(* CODESYS project code-dry-martini.project

Project tree, tasks and I/O mapping:
  Device : CODESYS Control Win V3, 3S - Smart Software Solutions GmbH, order no. 305021, version 3.5.6.10
    application Application
      libraries: Standard, * (System)
      task MainTask (cyclic, interval t#25ms, priority 1) calls PLC_PRG, Controller
      task Secondary_Tasks (cyclic, interval t#50ms, priority 2) calls Batelada, Envase, Descartar
      task Simulacao (cyclic, interval t#100ms, priority 1) calls SimulaContadores, SimulaSensores
      task PWM (cyclic, interval t#50ms, priority 1) calls pwmpou
      program PLC_PRG [LD]
      global variables Globals
      program Batelada [SFC]: ACT1_add_gin_and_vermouth, ACT2_stop_adding_vermouth, ACT3_stop_adding_start_mixing, ACT4_stop_cooling, ACT5_stop_mixing, ACT6_close107, ACT7_finish_transfer, Step10_entry, ACT12_LSHH, ACT13_start_transfer
      program Envase [SFC]: ACT8_start_engine, ACT9_stop_and_fill, ACT10_stop_filling, ACT14_setup_timers
      program SimulaSensores [ST]
      program SimulaContadores [ST]
      program Descartar [SFC]: Step0_entry, Step1_entry, Step2_entry, Step3_entry
      program Controller [SFC]: Init_entry
      trace PWM (task MainTask): LIGA_MOTOR, M101
      program pwmpou [SFC]: ACT15_time_control, ACT16_on, ACT17_off
      Symbols
*)

// Device/Application/Globals
VAR_GLOBAL
	// ATUADORES
	FCV101: BOOL := 0;
	FCV102: BOOL := 0;
	FCV103: BOOL := 0;
	FCV104: BOOL := 0;
	FCV105: BOOL := 0;
	FCV106: BOOL := 0;
	FCV107: BOOL := 0;
	BA101: BOOL := 0;
	FCV201: BOOL := 0;
	M101: BOOL := 0;
	M201: BOOL := 0;
	
	// SENSORES
	TSL101: BOOL := 0;
	LSL101: BOOL := 0;
	LSL102: BOOL := 0;
	LSH101: BOOL := 0;
	LSH102: BOOL := 0;
	LSL201: BOOL := 0;
	FV201: BOOL := 0;
	ZY201: BOOL := 0;
	ZY202: BOOL := 0;
	LSH201: BOOL := 0;
	LSHH201: BOOL := 0;
	
	// VARIAVEIS DE CONTROLE
	LigaAux: BOOL := 0;
	Emg: BOOL := 0;
	Auto: BOOL := 0;
	TempRM01: REAL := 25;
	TempAmbienteCelsius: REAL := 25;
	CapacidadeJA01: REAL := 15;
	Alert_TR01Empty: BOOL := 0;
	LIGA_MOTOR: BOOL := 0;
	
	//CONTADORES
	FQ101: REAL := 0; 
	FQ102: REAL := 0;
	FQ103: REAL := 0;
	FQ201: REAL := 0;
	RM01: REAL := 0;
	TP01: REAL := 0;
	JA01: REAL := 0;
	nBarril: INT := 0;
	
	// TIMERS
	tZY202: REAL := 0;
	tZY201: REAL := 0;
	
	ALARM3: BOOL := FALSE;
END_VAR

// Device/Application/PLC_PRG
PROGRAM PLC_PRG
VAR
	Liga: BOOL;
	// Emg: é global
	// Auto: é global
	Man: BOOL;
END_VAR

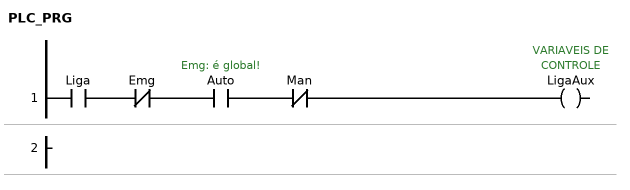
// NETWORK 1
//   Auto: Emg: é global!
//   LigaAux: VARIAVEIS DE CONTROLE
LigaAux := Liga AND NOT Emg AND Auto AND NOT Man;

// NETWORK 2

END_PROGRAM

// Device/Application/Controller
PROGRAM Controller
VAR
END_VAR

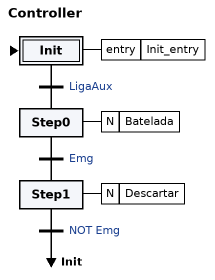
INITIAL_STEP Init:
    Init_entry(P1);  // entry action
END_STEP
TRANSITION FROM Init TO Step0
    := LigaAux;
END_TRANSITION
STEP Step0:
    Batelada(N);
END_STEP
TRANSITION FROM Step0 TO Step1
    := Emg;
END_TRANSITION
STEP Step1:
    Descartar(N);
END_STEP
TRANSITION FROM Step1 TO Init
    := NOT Emg;
END_TRANSITION

ACTION Init_entry:
TempAmbienteCelsius := 25;
CapacidadeJA01 := 15;
TempRM01:=TempAmbienteCelsius;
END_ACTION

END_PROGRAM

// Device/Application/Batelada
PROGRAM Batelada
VAR
END_VAR

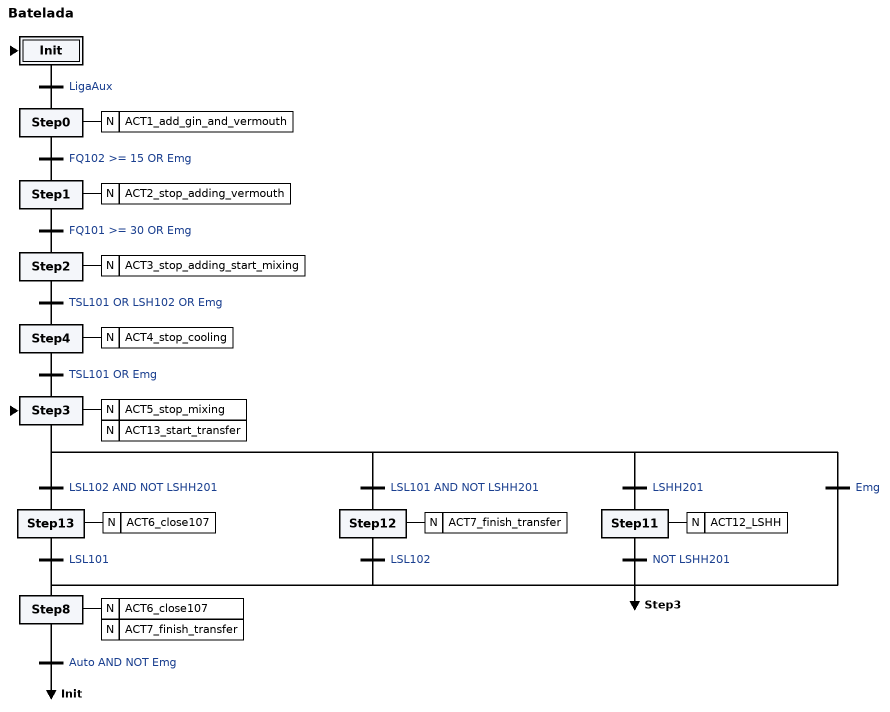
INITIAL_STEP Init:
END_STEP
TRANSITION FROM Init TO Step0
    := LigaAux;
END_TRANSITION
STEP Step0:
    ACT1_add_gin_and_vermouth(N);
END_STEP
TRANSITION FROM Step0 TO Step1
    := FQ102 >= 15 OR Emg;
END_TRANSITION
STEP Step1:
    ACT2_stop_adding_vermouth(N);
END_STEP
TRANSITION FROM Step1 TO Step2
    := FQ101 >= 30 OR Emg;
END_TRANSITION
STEP Step2:
    ACT3_stop_adding_start_mixing(N);
END_STEP
TRANSITION FROM Step2 TO Step4
    := TSL101 OR LSH102 OR Emg;
END_TRANSITION
STEP Step4:
    ACT4_stop_cooling(N);
END_STEP
TRANSITION FROM Step4 TO Step3
    := TSL101 OR Emg;
END_TRANSITION
STEP Step3:
    ACT5_stop_mixing(N);
    ACT13_start_transfer(N);
END_STEP
TRANSITION FROM Step3 TO Step13
    := LSL102 AND NOT LSHH201;
END_TRANSITION
STEP Step13:
    ACT6_close107(N);
END_STEP
TRANSITION FROM Step13 TO Step8
    := LSL101;
END_TRANSITION
TRANSITION FROM Step3 TO Step12
    := LSL101 AND NOT LSHH201;
END_TRANSITION
STEP Step12:
    ACT7_finish_transfer(N);
END_STEP
TRANSITION FROM Step12 TO Step8
    := LSL102;
END_TRANSITION
TRANSITION FROM Step3 TO Step11
    := LSHH201;
END_TRANSITION
STEP Step11:
    ACT12_LSHH(N);
END_STEP
TRANSITION FROM Step11 TO Step3
    := NOT LSHH201;
END_TRANSITION
TRANSITION FROM Step3 TO Step8
    := Emg;
END_TRANSITION
STEP Step8:
    ACT6_close107(N);
    ACT7_finish_transfer(N);
END_STEP
TRANSITION FROM Step8 TO Init
    := Auto AND NOT Emg;
END_TRANSITION

ACTION ACT1_add_gin_and_vermouth:
FCV101:=TRUE;
FCV102:=TRUE;
END_ACTION

ACTION ACT2_stop_adding_vermouth:
FCV102:=FALSE;
END_ACTION

ACTION ACT3_stop_adding_start_mixing:
FCV101:=FALSE;
LIGA_MOTOR:=TRUE;
FCV103:=TRUE;
END_ACTION

ACTION ACT4_stop_cooling:
FCV103:=FALSE;
END_ACTION

ACTION ACT5_stop_mixing:
LIGA_MOTOR:=FALSE;
END_ACTION

ACTION ACT6_close107:
FCV107:=FALSE;
END_ACTION

ACTION ACT7_finish_transfer:
FCV104:=FALSE;
FCV105:=FALSE;
BA101:=FALSE;
END_ACTION

ACTION Step10_entry:
FCV107:=TRUE;
FCV104:=TRUE;
FCV105:=TRUE;
BA101:=TRUE;
END_ACTION

ACTION ACT12_LSHH:
FCV104:=FALSE;
FCV105:=FALSE;
BA101:=FALSE;

IF TP01 <= 95 THEN
	LSHH201 := FALSE;
END_IF
END_ACTION

ACTION ACT13_start_transfer:
FCV107:=TRUE;
FCV104:=TRUE;
FCV105:=TRUE;
BA101:=TRUE;
END_ACTION

END_PROGRAM

// Device/Application/Envase
PROGRAM Envase
VAR
END_VAR

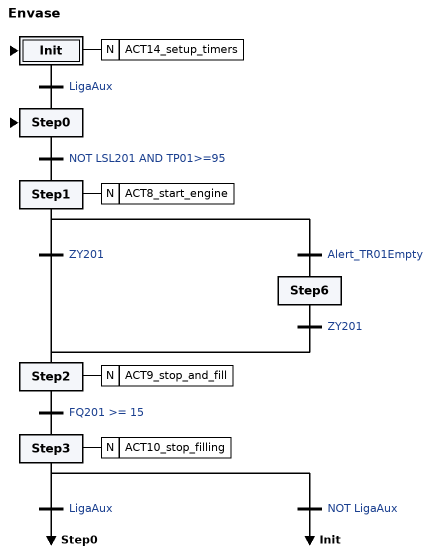
INITIAL_STEP Init:
    ACT14_setup_timers(N);
END_STEP
TRANSITION FROM Init TO Step0
    := LigaAux;
END_TRANSITION
STEP Step0:
END_STEP
TRANSITION FROM Step0 TO Step1
    := NOT LSL201 AND TP01>=95;
END_TRANSITION
STEP Step1:
    ACT8_start_engine(N);
END_STEP
TRANSITION FROM Step1 TO Step2
    := ZY201;
END_TRANSITION
TRANSITION FROM Step1 TO Step6
    := Alert_TR01Empty;
END_TRANSITION
STEP Step6:
END_STEP
TRANSITION FROM Step6 TO Step2
    := ZY201;
END_TRANSITION
STEP Step2:
    ACT9_stop_and_fill(N);
END_STEP
TRANSITION FROM Step2 TO Step3
    := FQ201 >= 15;
END_TRANSITION
STEP Step3:
    ACT10_stop_filling(N);
END_STEP
TRANSITION FROM Step3 TO Step0
    := LigaAux;
END_TRANSITION
TRANSITION FROM Step3 TO Init
    := NOT LigaAux;
END_TRANSITION

ACTION ACT8_start_engine:
M201:=TRUE;
END_ACTION

ACTION ACT9_stop_and_fill:
M201:=FALSE;
FCV201:=TRUE;
IF(Step2.t = T#15MS) THEN	
	ALARM3:=TRUE;
END_IF;
END_ACTION

ACTION ACT10_stop_filling:
FCV201:=FALSE;
END_ACTION

ACTION ACT14_setup_timers:
tZY202:=0;
tZY201:=0;
nBarril:=0;
END_ACTION

END_PROGRAM

// Device/Application/Descartar
PROGRAM Descartar
VAR
END_VAR

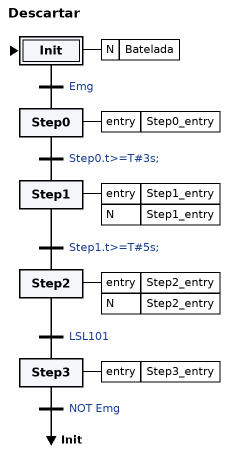
INITIAL_STEP Init:
    Batelada(N);
END_STEP
TRANSITION FROM Init TO Step0
    := Emg;
END_TRANSITION
STEP Step0:
    Step0_entry(P1);  // entry action
END_STEP
TRANSITION FROM Step0 TO Step1
    := Step0.t>=T#3s;
END_TRANSITION
STEP Step1:
    Step1_entry(P1);  // entry action
    Step1_entry(N);
END_STEP
TRANSITION FROM Step1 TO Step2
    := Step1.t>=T#5s;
END_TRANSITION
STEP Step2:
    Step2_entry(P1);  // entry action
    Step2_entry(N);
END_STEP
TRANSITION FROM Step2 TO Step3
    := LSL101;
END_TRANSITION
STEP Step3:
    Step3_entry(P1);  // entry action
END_STEP
TRANSITION FROM Step3 TO Init
    := NOT Emg;
END_TRANSITION

ACTION Step0_entry:
FCV101:=FALSE;
FCV102:=FALSE;
FCV103:=FALSE;
LIGA_MOTOR:=FALSE;
END_ACTION

ACTION Step1_entry:
FCV104:=TRUE;
FCV106:=TRUE;
BA101:=FALSE;
END_ACTION

ACTION Step2_entry:
BA101:=TRUE;
END_ACTION

ACTION Step3_entry:
BA101:=FALSE;
FCV104:=FALSE;
FCV105:=FALSE;
FCV106:=FALSE;
FCV107:=FALSE;
END_ACTION

END_PROGRAM

// Device/Application/SimulaContadores
PROGRAM SimulaContadores
VAR
	CapacidadeJaquetaRM01Litros: INT:=20; //capacidade em litros da jaqueta de resfriamento de RM01 (omisso na especificação)
	TempAmbienteCulsius: INT:= 25; //temperatura ambiente em celsius
	TOTALGIN: REAL:=0;
	TOTALVER: REAL:=0;
	TOTALDRY: REAL:=0;
//	LSL102: BOOL;
END_VAR

//ATENCAO: ESTE PROGRAMA RODA A CADA 100ms!

IF FCV101 THEN
	FQ101:=FQ101+0.6; // GIN 360 L/min = 6 L/s
	RM01:=RM01+0.6;
	TOTALGIN:=TOTALGIN+0.6;
	ELSE
		FQ101:=0;
END_IF

IF FCV102 THEN
	FQ102:=FQ102+0.5; // VERMOUTH 18 m³/h = 5 L/min
	RM01:=RM01+0.5;
	TOTALVER:=TOTALVER+0.5;
	ELSE
		FQ102:=0;
END_IF

IF FCV105 AND BA101 AND FCV104 THEN
	FQ103:=FQ103+1.5; // DRY MARTINI 54 m³/h = 15 L/min
	TP01:=TP01+1.5;
	TOTALDRY:=TOTALDRY+1.5;
ELSE
	IF NOT FCV105 THEN
		FQ103:=0;
	END_IF
END_IF

IF FCV104 AND RM01 > 0 THEN
	RM01:=RM01-1.5; 
END_IF

IF FCV201 AND TP01 > 0  THEN
	TP01:=TP01-0.3; // BICO INJETOR 10,8 m³/h = 3 L/s
	FQ201:=FQ201+0.3;
ELSE
	IF NOT FCV201 THEN
		FQ201:=0;
	END_IF
END_IF

//entrada de liquido refrigerante
IF (FCV103 AND (NOT LSH102)) THEN
	JA01:=JA01+0.5;
END_IF;

//saida de liquido refrigerante
IF (FCV107 AND (NOT LSL102)) THEN
	JA01:=JA01-0.5;
END_IF;

END_PROGRAM

// Device/Application/SimulaSensores
PROGRAM SimulaSensores
VAR
END_VAR

//ATENCAO: ESTE PROGRAMA RODA A CADA 100ms!

//sensor nivel BAIXO do Reator RM01
IF (RM01 <= 0) THEN
	RM01:=0;
	LSL101 := TRUE;
	TempRM01:=TempAmbienteCelsius; //caso reator esteja vazio, seta temperatura
	TSL101:=FALSE;
ELSE
	LSL101 := FALSE;
END_IF

//sensor nivel BAIXO jaqueta
IF (JA01 <= 0) THEN
	JA01:=0;
	LSL102:=TRUE;
ELSE
	LSL102:=FALSE;
END_IF;

//sensor nivel ALTO Jaqueta
IF (JA01 >= CapacidadeJA01) THEN
	LSH102:=TRUE;
ELSE
	LSH102:=FALSE;
END_IF;

// redução de temperatura provocada pela agitação
IF ( LIGA_MOTOR ) THEN
	IF TempRM01 > 0.1 THEN
		TSL101:=FALSE;
		TempRM01:=TempRM01-0.3;
	ELSE
		TSL101:=TRUE; // Termostato da jaqueta, ATIVA quando esta a 0 +- 1 graus
	END_IF;	
END_IF

// sensor nível ALTO e MUITO ALTO do tanque
IF TP01 >= 161.5 THEN
	LSH201 := TRUE;
	IF TP01 >= 180.5 THEN
		LSHH201 := TRUE;
	END_IF
ELSE 
	LSH201 := FALSE;
END_IF

// sensor nível BAIXO do tanque
IF TP01 <= 19 THEN
	LSL201 := 1;
ELSE 
	LSL201 := 0;
END_IF

//Timers da Esteira
IF M201 THEN 
	tZY201 := tZY201 + 0.1;
	tZY202 := tZY202 + 0.1;
END_IF

// IF NOT LSL201 THEN
//	tZY201 := tZY201 + 0.1;
// END_IF

//Simulador do sensor de barril no bico injetor
IF (tZY201 >= 5) THEN 
	ZY201 := TRUE;
ELSE 
	ZY201 := FALSE;	
END_IF

//Simulador de detectção de barril na saída
IF (tZY202 >= 3) THEN 
	ZY202 := TRUE;
ELSE 
	ZY202 := FALSE;
END_IF

IF ZY201 THEN // Reseta timer
	tZY201 := 0;
END_IF

IF ZY202 THEN //Contagem de Barris cheios
	nBarril := nBarril + 1;
	tZY202 := 0;
END_IF

IF tZY201 >= 15 THEN
	M201:=FALSE;
	Alert_TR01Empty:=TRUE;
END_IF

END_PROGRAM

// Device/Application/pwmpou
PROGRAM pwmpou
VAR
	time_on: TIME;
	time_off: TIME;
	motor_porcento_PWM: INT := 0;
END_VAR

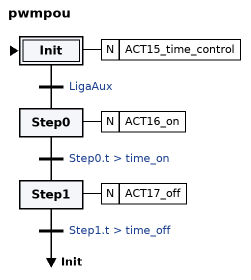
INITIAL_STEP Init:
    ACT15_time_control(N);
END_STEP
TRANSITION FROM Init TO Step0
    := LigaAux;
END_TRANSITION
STEP Step0:
    ACT16_on(N);
END_STEP
TRANSITION FROM Step0 TO Step1
    := Step0.t > time_on;
END_TRANSITION
STEP Step1:
    ACT17_off(N);
END_STEP
TRANSITION FROM Step1 TO Init
    := Step1.t > time_off;
END_TRANSITION

ACTION ACT15_time_control:
IF (LIGA_MOTOR AND motor_porcento_PWM < 100) THEN
	motor_porcento_PWM := motor_porcento_PWM+1;
ELSIF (motor_porcento_PWM > 0) THEN
	motor_porcento_PWM := motor_porcento_PWM-1;
END_IF
time_on := (T#50MS)*(motor_porcento_PWM/100);
time_off := (T#50MS)*((100-motor_porcento_PWM)/100);
END_ACTION

ACTION ACT16_on:
M101 := 1;
END_ACTION

ACTION ACT17_off:
M101 := 0;
END_ACTION

END_PROGRAM
